{attribute 'linkalways'} 
{attribute 'no_explicit_call' := 'This FB is a CLASS and must be accessed using methods or properties'}
{attribute 'enable_dynamic_creation'}
FUNCTION_BLOCK FINAL ADD_WORD EXTENDS Node
VAR
	in1 : _WORD(0);
	in2 : _WORD(0);
	out : _WORD(0);
END_VAR

METHOD PUBLIC Clone : I_Node
VAR
	pNode : POINTER TO ADD_WORD;
END_VAR
pNode := __NEW(ADD_WORD);
Clone := pNode^;
END_METHOD

METHOD FB_init : BOOL
VAR_INPUT
	bInitRetains : BOOL; // if TRUE, the retain variables are initialized (warm start / cold start)
	bInCopyCode : BOOL;  // if TRUE, the instance afterwards gets moved into the copy code (online change)
END_VAR
AddInput('in1',THIS^.in1);
AddInput('in2',THIS^.in2);
AddOutput('out', THIS^.out);
END_METHOD

METHOD PROTECTED OnExecute
VAR
END_VAR
out.Value := in1.Value + in2.Value;
END_METHOD

END_FUNCTION_BLOCK

(* stored: Version 1.1.0.1, ProductVersion 3.1.4024.15
   POU ADD_WORD: Id {f8e405b3-d781-45c2-b8c2-c8a13efdc00f}, SpecialFunc None
   Folder Constructor: Id {a011ac28-5fcd-4d8b-8b46-b5066a920456}
   Method Clone: Id {3cbde3f1-5a19-48b9-bfd3-0ae65df7ef47}
   Method FB_init: Id {36b3b274-2030-48f6-8a19-4937e7d0fec4}
   Method OnExecute: Id {7800ebaa-0666-43d9-8756-83251e805be8} *)
